(* CODESYS project mqttframework_11210.library
   Author: Filippo Boido
   Placeholder: MqttFramework
   Title: MqttFramework
   Version: 1.1.2.10
   Company: FactoryAutomation

Project tree, tasks and I/O mapping:
  libraries: StateMachineLib, * (FactoryAutomation); StepWorkerLib, * (FactoryAutomation); Tc2_Standard, * (Beckhoff Automation GmbH); Tc2_System, * (Beckhoff Automation GmbH); Tc2_Utilities, * (Beckhoff Automation GmbH); Tc3_Module, * (Beckhoff Automation GmbH)
  DUTs/
    data type E_AdsConnectorBusy
    data type E_MainStep
    data type ST_MqttAdsShell
    data type ST_MqttLifePackage
    type ST_MqttMessage [ST]
    data type ST_MqttPayload
  GVLs/
  POUs/
    program ADS [ST]
    function block AdsConnector [ST]: Busy, Error, Idle, Init, isConnected, Prepare, Ready, Waiting
    function block AdsSupplier [ST]
    function block MachineCycle [ST]: Busy, Error, Idle, Init, Prepare, Ready, Waiting
    program MAIN [ST]
    function block MqttClient [ST]: Busy, Error, Idle, Init, Prepare, Ready, Waiting, getNewMessage, isNewMessage, isPublishing, isSubscribing, publish, publishMessage, subscribe
  VISUs/
  program Version [ST]
*)

// DUTs/E_AdsConnectorBusy

TYPE E_AdsConnectorBusy :
(
	eNO_STEP := 0,
	eCHECK_IF_CONNECTED,
	eCONNECTED,
	eDISCONNECTED
)UINT;
END_TYPE

// DUTs/E_MainStep

TYPE E_MainStep :
(
	ePREPARE_SUBSCRIPTION := 0,
	ePREP_PUBLISH,
	ePUBLISH,
	eCHECK_SUBSCRIPTION,
	eEVAL_PAYLOAD,
	ePREPARE_PACKAGE_TIMER 
)UINT;
END_TYPE

// DUTs/ST_MqttAdsShell
{attribute 'pack_mode' := '1'}
TYPE ST_MqttAdsShell :
STRUCT
	bNewMessage : BOOL;
	sTopic : STRING(8);
	stMqttPayload : ST_MqttPayload;
END_STRUCT
END_TYPE

// DUTs/ST_MqttLifePackage
{attribute 'pack_mode' := '1'}
TYPE ST_MqttLifePackage :
STRUCT
	//State of the current machine
	uiStateMachine : UINT;
	dtDate : DATE_AND_TIME;
	sDateTime : STRING;
END_STRUCT
END_TYPE

// DUTs/ST_MqttPayload
{attribute 'pack_mode' := '1'}
TYPE ST_MqttPayload :
STRUCT
	id : UINT;
	data : ARRAY[1..32] OF Byte;
END_STRUCT
END_TYPE

// DUTs/ST_MqttMessage
{attribute 'pack_mode' := '1'}
TYPE ST_MqttMessage :
STRUCT
	sTopic : STRING;
	sMessage : T_MAXSTRING;
END_STRUCT
END_TYPE

// POUs/ADS
PROGRAM ADS
VAR
	fbAdsConnector : AdsConnector;
	fbMqttClient : MqttClient;
	sizeOfMqttPayload : UINT;
	sizeOfAdsShell : UINT;
	sizeOfTopic : UINT;
END_VAR

fbAdsConnector();
fbAdsConnector.Execute();
fbMqttClient();

sizeOfMqttPayload := SIZEOF(ST_MQTTPAYLOAD);
sizeOfAdsShell := SIZEOF(ST_MQTTADSSHELL);
sizeOfTopic := SIZEOF(ST_MQTTADSSHELL.sTopic);

END_PROGRAM

// POUs/AdsConnector
FUNCTION_BLOCK AdsConnector EXTENDS StateMachine
VAR_INPUT
END_VAR
VAR_OUTPUT
END_VAR
VAR
	fbStepWorkerBusy : FB_StepWorker;
	cbConnected : Boolean; //Custom Boolean
	fbAdsSupplier : AdsSupplier;
	
END_VAR

SUPER^();
Start();

METHOD PROTECTED Busy : BOOL
VAR_INPUT
END_VAR
VAR_INST
	eAdsConnectorBusy : E_AdsConnectorBusy;
END_VAR
eAdsConnectorBusy := fbStepWorkerBusy.getStep;
IF fbStepWorkerBusy.getStep = eNO_STEP 
THEN
	fbStepWorkerBusy.mNextStep(eCHECK_IF_CONNECTED);
END_IF


CASE fbStepWorkerBusy.getStep OF

	eCHECK_IF_CONNECTED:
	
		fbStepWorkerBusy.mAddCondition(cbConnected);
		fbStepWorkerBusy.mNextStep(eCONNECTED);
		
	eCONNECTED:
	
		fbAdsSupplier();
		IF NOT cbConnected.getValue
		THEN
			fbStepWorkerBusy.mNextStep(eDISCONNECTED);
		END_IF
	
	eDISCONNECTED:
	
		Done();
		fbStepWorkerBusy.mNextStep(eNO_STEP);
	
END_CASE
END_METHOD

METHOD PROTECTED  Error : BOOL
VAR_INPUT
END_VAR
END_METHOD

METHOD PROTECTED  Idle : BOOL
VAR_INPUT
END_VAR
END_METHOD

METHOD PROTECTED  Init : BOOL
VAR_INPUT
END_VAR
END_METHOD

PROPERTY isConnected : BOOL
GET
isConnected := cbConnected.getValue;
END_GET
END_PROPERTY

METHOD PROTECTED  Prepare : BOOL
VAR_INPUT
END_VAR
END_METHOD

METHOD PROTECTED  Ready : BOOL
VAR_INPUT
END_VAR
END_METHOD

METHOD PROTECTED  Waiting : BOOL
VAR_INPUT
END_VAR
END_METHOD

END_FUNCTION_BLOCK

// POUs/AdsSupplier
FUNCTION_BLOCK AdsSupplier
VAR_INPUT
	(* Here all mqtt packages that need to be exchanged.*)
END_VAR
VAR_OUTPUT
END_VAR
VAR
	
	fbLocalSystemTime : FB_LocalSystemTime := ( bEnable := TRUE, dwCycle := 1 );
	
	stMqttLifePackage : ST_MqttLifePackage;
	stEmptyLifePackage : ST_MqttLifePackage;
END_VAR

fbLocalSystemTime();
stMqttLifePackage := stEmptyLifePackage;
IF fbLocalSystemTime.bValid 
THEN
	stMqttLifePackage.uiStateMachine := MAIN.mainMachineCycle.eStateMachine;
	stMqttLifePackage.dtDate := SYSTEMTIME_TO_DT( fbLocalSystemTime.systemTime );
	stMqttLifePackage.sDateTime := DT_TO_STRING(stMqttLifePackage.dtDate);
END_IF

END_FUNCTION_BLOCK

// POUs/MAIN
PROGRAM MAIN 
VAR
	mainMachineCycle : MachineCycle;
	fbLifePackageTimer : TON := (PT := T#10S);
	fbStepWorker : FB_StepWorker;
	stMqttSubPayload : ST_MqttPayload;
	stMqttPubPayload : ST_MqttPayload;
	messageIndex : UINT;
	fbLocalSystemTime : FB_LocalSystemTime := ( bEnable := TRUE, dwCycle := 1 );
	udiTime : UDINT;
	udiReceivedTime : UDINT;
	//Zeitstempel der letzten Mqtt-Nachricht. Der Zeitstempel bezieht sich auf die Zeit kurz vor der Veröffentlichung.
	dtReceivedTime : DT;
END_VAR

mainMachineCycle();
fbLocalSystemTime();
(*Test your mqtt implementation here*)
fbLifePackageTimer();

CASE fbStepWorker.getStep OF

	ePREPARE_SUBSCRIPTION:
	
		IF ADS.fbAdsConnector.isConnected
		THEN
			IF ADS.fbMqttClient.Subscribe('TEST',ADR(MAIN))
			THEN
				
				fbStepWorker.mNextStep(ePREP_PUBLISH);
			END_IF
		END_IF
		
	ePREP_PUBLISH:	
	
		udiTime := DT_TO_UDINT(SYSTEMTIME_TO_DT(fbLocalSystemTIme.systemTime));
		stMqttPubPayload.id := stMqttPubPayload.id + 1;
		MEMCPY(ADR(stMqttPubPayload.data),ADR(udiTime),4);
		fbStepWorker.mNextStep(ePUBLISH);
		
	ePUBLISH:
		
		IF ADS.fbMqttClient.Publish('TEST',stMqttPubPayload,ADR(MAIN))
		THEN
			fbStepWorker.mNextStep(eCHECK_SUBSCRIPTION);
		END_IF	
			
	eCHECK_SUBSCRIPTION:
		
		messageIndex := ADS.fbMqttClient.isNewMessage('TEST');
		IF messageIndex > 0
		THEN
			stMqttSubPayload := Ads.fbMqttClient.getNewMessage(messageIndex);
			fbStepWorker.mNextStep(eEVAL_PAYLOAD);
		END_IF
			
	eEVAL_PAYLOAD:
	
		//last received time via mqtt
		MEMCPY(ADR(udiReceivedTime),ADR(stMqttSubPayload.data),4);
		dtReceivedTime := UDINT_TO_DT(udiReceivedTime);
		fbLifePackageTimer.IN := TRUE;
		IF fbLifePackageTimer.Q
			AND fbLocalSystemTime.bValid
		THEN
			fbLifePackageTimer.IN := FALSE;
			fbStepWorker.mNextStep(ePREP_PUBLISH);
		END_IF
		
	
END_CASE

END_PROGRAM

// POUs/MachineCycle
FUNCTION_BLOCK MachineCycle EXTENDS StateMachine
VAR_INPUT
END_VAR
VAR_OUTPUT
END_VAR
VAR
END_VAR

SUPER^();
Start();

METHOD PROTECTED Busy : BOOL
VAR_INPUT
END_VAR
VAR_INST
	eAdsConnectorBusy : E_AdsConnectorBusy;
END_VAR
END_METHOD

METHOD PROTECTED  Error : BOOL
VAR_INPUT
END_VAR
END_METHOD

METHOD PROTECTED  Idle : BOOL
VAR_INPUT
END_VAR
END_METHOD

METHOD PROTECTED  Init : BOOL
VAR_INPUT
END_VAR
END_METHOD

METHOD PROTECTED  Prepare : BOOL
VAR_INPUT
END_VAR
END_METHOD

METHOD PROTECTED  Ready : BOOL
VAR_INPUT
END_VAR
(*
Check conditions to fire Execute() here and put the StateMachine in Busy mode
*)
END_METHOD

METHOD PROTECTED  Waiting : BOOL
VAR_INPUT
END_VAR
END_METHOD

END_FUNCTION_BLOCK

// POUs/MqttClient
FUNCTION_BLOCK MqttClient EXTENDS StateMachine
VAR_INPUT
END_VAR
VAR_OUTPUT
	
END_VAR

VAR
	bPublishing : BOOL;
	bPublished : BOOL;
	bSubscribing : BOOL;
	bSubscribed : BOOL;
	bPublishingMessage : BOOL;
	bPublishedMessage : BOOL;
	uiSubscriptionCounter : UINT := 1;
	uiPublicationCounter : UINT := 1;
	uiMessageCounter : UINT := 0;
	
	uiSizeOfSubscriptions : UINT;
	uiSizeOfPublications : UINT;
	
	aAdsSubscriptionStorage : ARRAY[1..cMaxSubscriptions] OF ST_MqttAdsShell;
	
	aAdsPublicationStorage : ARRAY[1..cMaxPublications] OF ST_MqttAdsShell;
	aAdsOldPublications : ARRAY[1..cMaxPublications] OF ST_MqttAdsShell;
	
	
	aAdsMessageStorage : ARRAY[1..cMaxMessages] OF ST_MqttMessage;
	aAdsOldMessages : ARRAY[1..cMaxMessages] OF ST_MqttMessage;
	
	sizeOfAdsShell : UINT;
	
	i : UINT;
	pvLockPublish : PVOID;
	pvLockSubscribe : PVOID;
END_VAR

VAR CONSTANT
	cMaxSubscriptions : UINT := 10;
	cMaxPublications : UINT := 10;
	cMaxMessages : UINT := 10;
END_VAR

SUPER^();
Start();

METHOD PROTECTED Busy : BOOL
VAR_INPUT
END_VAR
VAR_INST
	eAdsConnectorBusy : E_AdsConnectorBusy;
END_VAR
END_METHOD

METHOD PROTECTED  Error : BOOL
VAR_INPUT
END_VAR
END_METHOD

METHOD PROTECTED  Idle : BOOL
VAR_INPUT
END_VAR
END_METHOD

METHOD PROTECTED  Init : BOOL
VAR_INPUT
END_VAR
uiSizeOfSubscriptions := SIZEOF(aAdsSubscriptionStorage);
uiSizeOfPublications := SIZEOF(aAdsPublicationStorage);

sizeOfAdsShell := SIZEOF(ST_MQTTADSSHELL);
END_METHOD

METHOD PROTECTED  Prepare : BOOL
VAR_INPUT
END_VAR
END_METHOD

METHOD PROTECTED  Ready : BOOL
VAR_INPUT
END_VAR
(*
Check conditions to fire Execute() here and put the StateMachine in Busy mode
*)
END_METHOD

METHOD PROTECTED  Waiting : BOOL
VAR_INPUT
END_VAR
END_METHOD

METHOD getNewMessage : ST_MqttPayload
VAR_INPUT
	index : UINT;
END_VAR
VAR
	stEmptyMqttPayload : ST_MqttPayload;
END_VAR
IF index > 0
	AND index <= cMaxSubscriptions 
THEN
	aAdsSubscriptionStorage[index].bNewMessage := FALSE;
	getNewMessage := aAdsSubscriptionStorage[index].stMqttPayload;
	aAdsSubscriptionStorage[index].stMqttPayload := stEmptyMqttPayload;
END_IF
END_METHOD

METHOD isNewMessage : UINT
VAR_INPUT
	sTopic : STRING(8);
END_VAR
VAR
	i : UINT;
END_VAR
FOR i := 1 TO cMaxSubscriptions
DO
	IF aAdsSubscriptionStorage[i].sTopic = sTopic 
		AND_THEN aAdsSubscriptionStorage[i].bNewMessage
	THEN
		isNewMessage := i;
		RETURN;
	END_IF
	
END_FOR
END_METHOD

METHOD isPublishing : BOOL
VAR_INPUT
END_VAR
isPublishing := bPublishing;
END_METHOD

METHOD isSubscribing : BOOL
VAR_INPUT
END_VAR
isSubscribing := bSubscribing;
END_METHOD

METHOD publish : BOOL //Return true if published
VAR_INPUT
	sTopic : STRING(8);
	stMqttPayload : ST_MqttPayload;
	pvLock : PVOID;
END_VAR

VAR
	aEmptyPublicationStorage : ARRAY[1..cMaxPublications] OF ST_MqttAdsShell;
	
END_VAR
IF  (	bPublishing
		AND NOT bPublished)
	OR 
	(	bPublishing 
		AND bPublished
		AND THIS^.pvLockPublish <> pvLock)		
THEN

	RETURN;
	
ELSIF 	bPublishing 
	AND bPublished
	AND THIS^.pvLockPublish = pvLock
THEN

	bPublishing := FALSE;
	bPublished := FALSE;
	Publish := TRUE;
	RETURN;
	
ELSIF 	NOT bPublishing
	AND NOT bPublished
THEN
 
	THIS^.pvLockPublish := pvLock;
	bPublishing := TRUE;
	
END_IF

IF uiPublicationCounter > cMaxPublications
THEN
	aAdsOldPublications := aAdsPublicationStorage;
	aAdsPublicationStorage := aEmptyPublicationStorage;	
	uiPublicationCounter := 1;
END_IF

aAdsPublicationStorage[uiPublicationCounter].stMqttPayload := stMqttPayload;
aAdsPublicationStorage[uiPublicationCounter].sTopic := sTopic;
uiPublicationCounter := uiPublicationCounter + 1;
END_METHOD

METHOD publishMessage : BOOL
VAR_INPUT
	sTopic : STRING(8);
	sMessage : T_MAXSTRING;
	pvLock : PVOID;
END_VAR

VAR
	aEmptyMessages : ARRAY[1..cMaxMessages] OF ST_MqttMessage;
END_VAR
IF  (	bPublishingMessage
		AND NOT bPublishedMessage)
	OR 
	(	bPublishingMessage 
		AND bPublishedMessage
		AND THIS^.pvLockPublish <> pvLock)		
THEN

	RETURN;
	
ELSIF 	bPublishingMessage 
	AND bPublishedMessage
	AND THIS^.pvLockPublish = pvLock
THEN

	bPublishingMessage := FALSE;
	bPublishedMessage := FALSE;
	publishMessage := TRUE;
	RETURN;
	
ELSIF 	NOT bPublishingMessage
	AND NOT bPublishedMessage
THEN
 
	THIS^.pvLockPublish := pvLock;
	bPublishingMessage := TRUE;
	
END_IF

IF uiMessageCounter >= cMaxMessages
THEN
	aAdsOldMessages := aAdsMessageStorage;
	aAdsMessageStorage := aEmptyMessages;	
	uiMessageCounter := 0;
END_IF

uiMessageCounter := uiMessageCounter + 1;
aAdsMessageStorage[uiMessageCounter].sMessage := sMessage;
aAdsMessageStorage[uiMessageCounter].sTopic := sTopic;
END_METHOD

METHOD subscribe : BOOL  //Return true if subscribed
VAR_INPUT
	sTopic : STRING(8);
	pvLock : POINTER TO PVOID;
END_VAR
IF 	uiSubscriptionCounter > cMaxSubscriptions
	OR
	(	bSubscribing = TRUE 
		AND bSubscribed = FALSE) 
	OR
	(	bSubscribing = TRUE
		AND bSubscribed = TRUE
		AND pvLockSubscribe <> pvLock)		
THEN

	RETURN;
	
ELSIF 	bSubscribing = TRUE
		AND bSubscribed = TRUE
		AND pvLockSubscribe = pvLock
THEN

	bSubscribing := FALSE;
	bSubscribed := FALSE;
	Subscribe := TRUE;
	
	RETURN;
	
ELSIF	bSubscribing = FALSE
		AND bSubscribed = FALSE
THEN

	bSubscribing := TRUE;
	pvLockSubscribe := pvLock;
	
END_IF

aAdsSubscriptionStorage[uiSubscriptionCounter].sTopic := sTopic;
uiSubscriptionCounter := uiSubscriptionCounter + 1;
END_METHOD

END_FUNCTION_BLOCK

// Version
PROGRAM Version
VAR
END_VAR

(*

1.0.1.1:	Boido	020120

Version.txt replaced with Version PRG

1.0.2.2:	Boido	020120

VersionLib removed.

1.0.3.3:	Boido	090220

Bugfix in MqttClient.getNewMessage();

1.0.4.4:	Boido	240520

Date and time as String in ST_MqttLifePackage

1.0.5.5:	Boido	300520

isPublishing and isSubscribing methods added to MqttClient

1.0.6.6:	Boido	300520

pvLockSubscribe and pvLockPublish added to MqttClient

1.0.7.7:	Boido	090620

changed E_MainStep and E_AdsConnectorBusy enum-type to UINT

1.1.0.8:	Boido	140620

Ability to send strings with publishMessage added to the mqttClient

1.1.1.9:	Boido 	150620

Bugfix array access in fbMqttClient.publishMessage()
Bugfix bPublishingMessage bPublishedMessage in fbMqttClient.publishMessage()

1.1.2.10:	Boido 	160620

uiMessageCounter in fbMqttClient.publishMessage() reset when it equals cMaxMessages

*)

END_PROGRAM
